{attribute 'qualified_only'}
TYPE E_DrivingPinSelection :
(
	Both,
    Left,
    Right
)USINT;
END_TYPE

(* stored: Version 1.1.0.1, ProductVersion 3.1.4024.11
   DUT E_DrivingPinSelection: Id {049b60a3-f80a-4e49-a654-6c34f74569cd} *)
